// TIA Portal V20 export
TYPE "UDT_EventosPantalla"
   STRUCT
      Mckey : UDInt;
      NivelVisual : UInt;
      LineaTexto_01 : String[48];   // Primer Linea del Texto a Visulizar
      LineaTexto_02 : String[48];   // Segunda Linea del Texto a Visulizar
      LineaTexto_03 : String[48];   // Tercera Linea del Texto a Visulizar
      LineaTexto_04 : String[48];   // Cuarta Linea del Texto a Visulizar
   END_STRUCT;
END_TYPE
